# EPICS autosave request: iocBoot/gmca_23b_ioc2/dbSave/bluiceRuns.req
$(P)runCount
$(P)currentRun
$(P)isActive
$(P)doseMode
$(P)updated
